{attribute 'GeneratedUsingTerminal: EK1100-0000-0018'}
{attribute addProperty BoxType "EK1100-0000-0018"}
{attribute addProperty Id "Beckhoff_ELM31xxEK1122Beckhoff_ELM31xxEK1122_3373CF362A_0001_ELM3102_0000_0016ELM3102_73CCAB7A50A_0002_ELM3102_0000_0017ELM3102_73CCAB7A50A_0003_ELM3102_0000_0018ELM3102_73CCAB7A50A_0004_ELM3104_0000_0016ELM3104_7474644C72A_0005_ELM3104_0000_0017ELM3104_7474644C72A_0006_ELM3104_0000_0018ELM3104_7474644C72A_0007_ELM3142_0000_0016ELM3142_73CCAB7A50A_0008_ELM3142_0000_0017ELM3142_73CCAB7A50A_0009_ELM3144_0000_0016ELM3144_7474644C72A_0010_ELM3144_0000_0017ELM3144_7474644C72A_0011_ELM3146_0000_0016ELM3146_CCD8D99694A_0012_ELM3146_0000_0017ELM3146_CCD8D99694A_0013_ELM3146_0000_0018ELM3146_CCD8D99694A_0014_ELM3148_0000_0017ELM3148_BBE3CE2D116A_0015_ELM3148_0000_0018ELM3148_BBE3CE2D116A_0016_ELM3148_0000_0019ELM3148_BBE3CE2D116"}
{attribute addProperty CRC "2265058986"}
{attribute addProperty Size "1242"}
TYPE Beckhoff_ELM31xx_87020EAA EXTENDS EK1100_AB5A9467 :
STRUCT
	{attribute addProperty Name "Beckhoff_ELM31xxEK1122"}
	{attribute addProperty PreviousPort "Beckhoff ELM31xx : B"}
	Beckhoff_ELM31xxEK1122 : Beckhoff_ELM31xxEK1122_3373CF36;
	{attribute addProperty Name "A_0001_ELM3102_0000_0016"}
	{attribute addProperty PreviousPort "Beckhoff ELM31xxEK1122 : C"}
	A_0001_ELM3102_0000_0016 : ELM3102_73CCAB7A;
	{attribute addProperty Name "A_0002_ELM3102_0000_0017"}
	{attribute addProperty PreviousPort "A_0001(ELM3102-0000-0016) : B"}
	A_0002_ELM3102_0000_0017 : ELM3102_73CCAB7A;
	{attribute addProperty Name "A_0003_ELM3102_0000_0018"}
	{attribute addProperty PreviousPort "A_0002(ELM3102-0000-0017) : B"}
	A_0003_ELM3102_0000_0018 : ELM3102_73CCAB7A;
	{attribute addProperty Name "A_0004_ELM3104_0000_0016"}
	{attribute addProperty PreviousPort "A_0003(ELM3102-0000-0018) : B"}
	A_0004_ELM3104_0000_0016 : ELM3104_7474644C;
	{attribute addProperty Name "A_0005_ELM3104_0000_0017"}
	{attribute addProperty PreviousPort "A_0004(ELM3104-0000-0016) : B"}
	A_0005_ELM3104_0000_0017 : ELM3104_7474644C;
	{attribute addProperty Name "A_0006_ELM3104_0000_0018"}
	{attribute addProperty PreviousPort "A_0005(ELM3104-0000-0017) : B"}
	A_0006_ELM3104_0000_0018 : ELM3104_7474644C;
	{attribute addProperty Name "A_0007_ELM3142_0000_0016"}
	{attribute addProperty PreviousPort "A_0006(ELM3104-0000-0018) : B"}
	A_0007_ELM3142_0000_0016 : ELM3142_73CCAB7A;
	{attribute addProperty Name "A_0008_ELM3142_0000_0017"}
	{attribute addProperty PreviousPort "A_0007(ELM3142-0000-0016) : B"}
	A_0008_ELM3142_0000_0017 : ELM3142_73CCAB7A;
	{attribute addProperty Name "A_0009_ELM3144_0000_0016"}
	{attribute addProperty PreviousPort "A_0008(ELM3142-0000-0017) : B"}
	A_0009_ELM3144_0000_0016 : ELM3144_7474644C;
	{attribute addProperty Name "A_0010_ELM3144_0000_0017"}
	{attribute addProperty PreviousPort "A_0009(ELM3144-0000-0016) : B"}
	A_0010_ELM3144_0000_0017 : ELM3144_7474644C;
	{attribute addProperty Name "A_0011_ELM3146_0000_0016"}
	{attribute addProperty PreviousPort "A_0010(ELM3144-0000-0017) : B"}
	A_0011_ELM3146_0000_0016 : ELM3146_CCD8D996;
	{attribute addProperty Name "A_0012_ELM3146_0000_0017"}
	{attribute addProperty PreviousPort "A_0011(ELM3146-0000-0016) : B"}
	A_0012_ELM3146_0000_0017 : ELM3146_CCD8D996;
	{attribute addProperty Name "A_0013_ELM3146_0000_0018"}
	{attribute addProperty PreviousPort "A_0012(ELM3146-0000-0017) : B"}
	A_0013_ELM3146_0000_0018 : ELM3146_CCD8D996;
	{attribute addProperty Name "A_0014_ELM3148_0000_0017"}
	{attribute addProperty PreviousPort "A_0013(ELM3146-0000-0018) : B"}
	A_0014_ELM3148_0000_0017 : ELM3148_BBE3CE2D;
	{attribute addProperty Name "A_0015_ELM3148_0000_0018"}
	{attribute addProperty PreviousPort "A_0014(ELM3148-0000-0017) : B"}
	A_0015_ELM3148_0000_0018 : ELM3148_BBE3CE2D;
	{attribute addProperty Name "A_0016_ELM3148_0000_0019"}
	{attribute addProperty PreviousPort "A_0015(ELM3148-0000-0018) : B"}
	A_0016_ELM3148_0000_0019 : ELM3148_BBE3CE2D;
END_STRUCT
END_TYPE

(* stored: Version 1.2.0.0, ProductVersion 3.1.4024.9
   DUT Beckhoff_ELM31xx_87020EAA: Id {033ef3e5-bad5-45d1-91b5-1cf49b20c142} *)
